// TIA Portal V19 export
TYPE "LubrPump_Par"
// stored: Access Published
   STRUCT
      LowLevelCheckTime : Time;
      ValveONTime : Time;
      ValveOFFTime : Time;
   END_STRUCT;
END_TYPE
